// Checks if a string is an unsigned interger
FUNCTION F_ISUNSIGNEDINT : BOOL
VAR_INPUT
	sValue : REFERENCE TO STRING;
END_VAR
VAR
	i : T_Size;
END_VAR

F_TRIMWHITESPACE(sValue, T_Whitespace_Location.Both);

IF NOT F_ISDIGIT(F_BYTETOCHAR(sValue[0])) THEN RETURN; END_IF
WHILE F_ISDIGIT(F_BYTETOCHAR(sValue[i])) DO i := i + 1; END_WHILE
F_ISUNSIGNEDINT := sValue[i] = 0;

END_FUNCTION

(* stored: Version 1.1.0.1, ProductVersion 3.1.4024.4
   POU F_ISUNSIGNEDINT: Id {e25af886-1eea-4141-8cc6-330bf17a78ea}, SpecialFunc None *)
